RoboDK station: robodkproject048037074.rdk

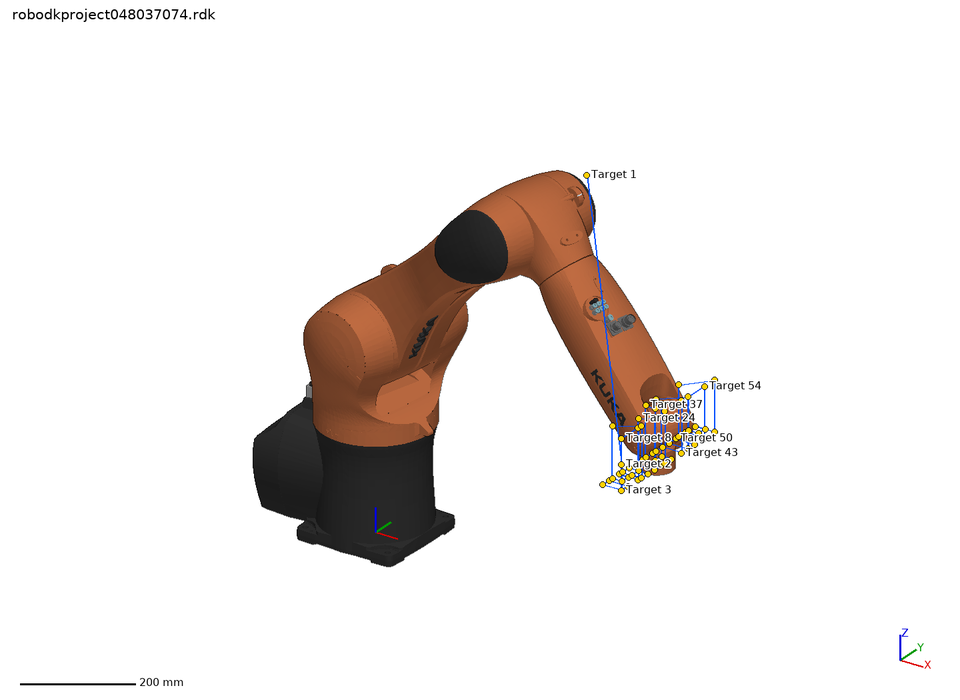
[picture v0: the station drawn from its stored meshes, robots at their saved joint values, targets as dots, program paths as lines]
Station robodkproject048037074 (saved by RoboDK 5.9.4). Poses are relative to the parent item; angles as X-Y-Z fixed-axis rotations.
  - frame KUKA KR 6 R900 sixx Base at (0, 0, 0) mm
    - robot KUKA KR 6 R900 sixx: 6 axes, payload 6 kg, reach 901 mm, repeatability 0.03 mm, weight 52 kg
        modified DH rows (alpha deg, a mm, theta deg, d mm): 0, 0, 0, 400; -90, 25, 0, 0; 0, 455, -90, 0; -90, 35, 0, 420; 90, 0, 0, 0; -90, 0, 180, 80
        joint limits [-170, -190, -120, -185, -120, -350] to [170, 45, 156, 185, 120, 350]; home [0, -90, 90, 0, 0, 0]; saved at [8.973, -42.929, 89.308, 0, 43.621, 8.973]
    - target Target 1 (Cartesian target) at (445, 0, 810) mm, rotated rx 180 ry 0 rz -180 deg; joints [0, -90, 90, 0, 90, 0] of KUKA KR 6 R900 sixx
    - target Target 2 (Cartesian target) at (665, -210, 400) mm, rotated rx 180 ry 0 rz -180 deg; joints [17.526, -44.432, 83.664, 0, 50.767, 17.526] of KUKA KR 6 R900 sixx
    - target Target 3 (Cartesian target) at (665, -210, 350) mm, rotated rx 180 ry 0 rz 180 deg; joints [17.526, -40.592, 84.501, 0, 46.092, 17.526] of KUKA KR 6 R900 sixx
    - target Target 4 (Cartesian target) at (625, -210, 350) mm, rotated rx 180 ry 0 rz -180 deg; joints [18.572, -44.227, 91.979, 0, 42.249, 18.572] of KUKA KR 6 R900 sixx
    - target Target 5 (Cartesian target) at (625, -190, 350) mm, rotated rx 180 ry 0 rz -180 deg; joints [16.909, -44.787, 93.129, 0, 41.657, 16.909] of KUKA KR 6 R900 sixx
    - target Target 6 (Cartesian target) at (665, -190, 350) mm, rotated rx 180 ry 0 rz -180 deg; joints [15.945, -41.161, 85.669, 0, 45.491, 15.945] of KUKA KR 6 R900 sixx
    - target Target 7 (Cartesian target) at (665, -210, 350) mm, rotated rx 180 ry 0 rz 180 deg; joints [17.526, -40.592, 84.501, 0, 46.092, 17.526] of KUKA KR 6 R900 sixx
    - target Target 8 (Cartesian target) at (665, -210, 450) mm, rotated rx 180 ry 0 rz 180 deg; joints [17.526, -47.839, 82.061, 0, 55.777, 17.526] of KUKA KR 6 R900 sixx
    - target Target 9 (Cartesian target) at (665, -160, 450) mm, rotated rx 180 ry 0 rz -180 deg; joints [13.528, -49.327, 84.778, 0, 54.549, 13.528] of KUKA KR 6 R900 sixx
    - target Target 10 (Cartesian target) at (665, -160, 350) mm, rotated rx 180 ry 0 rz -180 deg; joints [13.528, -41.903, 87.197, 0, 44.706, 13.528] of KUKA KR 6 R900 sixx
    - target Target 11 (Cartesian target) at (625, -160, 350) mm, rotated rx 180 ry 0 rz -180 deg; joints [14.359, -45.52, 94.638, 0, 40.882, 14.359] of KUKA KR 6 R900 sixx
    - target Target 12 (Cartesian target) at (645, -160, 350) mm, rotated rx 180 ry 0 rz -180 deg; joints [13.932, -43.745, 90.985, 0, 42.759, 13.932] of KUKA KR 6 R900 sixx
    - target Target 13 (Cartesian target) at (645, -180, 350) mm, rotated rx 180 ry 0 rz -180 deg; joints [15.593, -43.268, 90.005, 0, 43.263, 15.593] of KUKA KR 6 R900 sixx
    - target Target 14 (Cartesian target) at (625, -180, 350) mm, rotated rx 180 ry 0 rz -180 deg; joints [16.066, -45.045, 93.661, 0, 41.384, 16.066] of KUKA KR 6 R900 sixx
    - target Target 15 (Cartesian target) at (625, -180, 450) mm, rotated rx 180 ry 0 rz -180 deg; joints [16.066, -52.933, 91.269, 0, 51.664, 16.066] of KUKA KR 6 R900 sixx
    - target Target 16 (Cartesian target) at (665, -150, 450) mm, rotated rx 180 ry 0 rz -180 deg; joints [12.711, -49.576, 85.231, 0, 54.345, 12.711] of KUKA KR 6 R900 sixx
    - target Target 17 (Cartesian target) at (665, -150, 350) mm, rotated rx 180 ry 0 rz -180 deg; joints [12.711, -42.122, 87.647, 0, 44.475, 12.711] of KUKA KR 6 R900 sixx
    - target Target 18 (Cartesian target) at (665, -130, 350) mm, rotated rx 180 ry 0 rz -180 deg; joints [11.061, -42.516, 88.458, 0, 44.058, 11.061] of KUKA KR 6 R900 sixx
    - target Target 19 (Cartesian target) at (625, -130, 350) mm, rotated rx 180 ry 0 rz 180 deg; joints [11.75, -46.127, 95.887, 0, 40.24, 11.75] of KUKA KR 6 R900 sixx
    - target Target 20 (Cartesian target) at (625, -150, 350) mm, rotated rx 180 ry 0 rz -180 deg; joints [13.496, -45.736, 95.083, 0, 40.653, 13.496] of KUKA KR 6 R900 sixx
    - target Target 21 (Cartesian target) at (665, -150, 350) mm, rotated rx 180 ry 0 rz -180 deg; joints [12.711, -42.122, 87.647, 0, 44.475, 12.711] of KUKA KR 6 R900 sixx
    - target Target 22 (Cartesian target) at (645, -150, 350) mm, rotated rx 180 ry 0 rz -180 deg; joints [13.092, -43.962, 91.432, 0, 42.53, 13.092] of KUKA KR 6 R900 sixx
    - target Target 23 (Cartesian target) at (645, -130, 350) mm, rotated rx 180 ry 0 rz -180 deg; joints [11.395, -44.353, 92.238, 0, 42.115, 11.395] of KUKA KR 6 R900 sixx
    - target Target 24 (Cartesian target) at (645, -130, 450) mm, rotated rx 180 ry 0 rz -180 deg; joints [11.395, -52.134, 89.842, 0, 52.292, 11.395] of KUKA KR 6 R900 sixx
    - target Target 25 (Cartesian target) at (665, -110, 450) mm, rotated rx 180 ry 0 rz -180 deg; joints [9.392, -50.412, 86.745, 0, 53.667, 9.392] of KUKA KR 6 R900 sixx
    - target Target 26 (Cartesian target) at (665, -110, 350) mm, rotated rx 180 ry 0 rz -180 deg; joints [9.392, -42.854, 89.153, 0, 43.701, 9.392] of KUKA KR 6 R900 sixx
    - target Target 27 (Cartesian target) at (665, -90, 350) mm, rotated rx 180 ry 0 rz -180 deg; joints [7.707, -43.135, 89.731, 0, 43.404, 7.707] of KUKA KR 6 R900 sixx
    - target Target 28 (Cartesian target) at (625, -90, 350) mm, rotated rx 180 ry 0 rz -180 deg; joints [8.194, -46.74, 97.15, 0, 39.59, 8.194] of KUKA KR 6 R900 sixx
    - target Target 29 (Cartesian target) at (625, -110, 350) mm, rotated rx 180 ry 0 rz -180 deg; joints [9.982, -46.461, 96.576, 0, 39.885, 9.982] of KUKA KR 6 R900 sixx
    - target Target 30 (Cartesian target) at (665, -110, 350) mm, rotated rx 180 ry 0 rz -180 deg; joints [9.392, -42.854, 89.153, 0, 43.701, 9.392] of KUKA KR 6 R900 sixx
    - target Target 31 (Cartesian target) at (665, -110, 450) mm, rotated rx 180 ry 0 rz -180 deg; joints [9.392, -50.412, 86.745, 0, 53.667, 9.392] of KUKA KR 6 R900 sixx
    - target Target 32 (Cartesian target) at (665, -80, 450) mm, rotated rx 180 ry 0 rz -180 deg; joints [6.86, -50.87, 87.572, 0, 53.298, 6.86] of KUKA KR 6 R900 sixx
    - target Target 33 (Cartesian target) at (665, -80, 350) mm, rotated rx 180 ry 0 rz -180 deg; joints [6.86, -43.254, 89.976, 0, 43.278, 6.86] of KUKA KR 6 R900 sixx
    - target Target 34 (Cartesian target) at (665, -60, 350) mm, rotated rx 180 ry 0 rz -180 deg; joints [5.156, -43.45, 90.38, 0, 43.07, 5.156] of KUKA KR 6 R900 sixx
    - target Target 35 (Cartesian target) at (625, -60, 350) mm, rotated rx 180 ry 0 rz -180 deg; joints [5.484, -47.054, 97.797, 0, 39.258, 5.484] of KUKA KR 6 R900 sixx
    - target Target 36 (Cartesian target) at (625, -80, 350) mm, rotated rx 180 ry 0 rz -180 deg; joints [7.294, -46.859, 97.395, 0, 39.464, 7.294] of KUKA KR 6 R900 sixx
    - target Target 37 (Cartesian target) at (625, -80, 450) mm, rotated rx 180 ry 0 rz -180 deg; joints [7.294, -55.044, 95.003, 0, 50.041, 7.294] of KUKA KR 6 R900 sixx
    - target Target 38 (Cartesian target) at (645, -80, 450) mm, rotated rx 180 ry 0 rz -180 deg; joints [7.07, -52.982, 91.355, 0, 51.626, 7.07] of KUKA KR 6 R900 sixx
    - target Target 39 (Cartesian target) at (645, -80, 350) mm, rotated rx 180 ry 0 rz -180 deg; joints [7.07, -45.087, 93.747, 0, 41.34, 7.07] of KUKA KR 6 R900 sixx
    - target Target 40 (Cartesian target) at (645, -60, 350) mm, rotated rx 180 ry 0 rz -180 deg; joints [5.315, -45.282, 94.15, 0, 41.133, 5.315] of KUKA KR 6 R900 sixx
    - target Target 41 (Cartesian target) at (645, -60, 450) mm, rotated rx 180 ry 0 rz -180 deg; joints [5.315, -53.208, 91.758, 0, 51.45, 5.315] of KUKA KR 6 R900 sixx
    - target Target 42 (Cartesian target) at (665, -30, 450) mm, rotated rx 180 ry 0 rz -180 deg; joints [2.583, -51.313, 88.369, 0, 52.944, 2.583] of KUKA KR 6 R900 sixx
    - target Target 43 (Cartesian target) at (665, -30, 350) mm, rotated rx 180 ry 0 rz -180 deg; joints [2.583, -43.64, 90.769, 0, 42.87, 2.583] of KUKA KR 6 R900 sixx
    - target Target 44 (Cartesian target) at (625, -30, 350) mm, rotated rx 180 ry 0 rz -180 deg; joints [2.748, -47.243, 98.185, 0, 39.058, 2.748] of KUKA KR 6 R900 sixx
    - target Target 45 (Cartesian target) at (625, -50, 350) mm, rotated rx 180 ry 0 rz -180 deg; joints [4.574, -47.131, 97.955, 0, 39.176, 4.574] of KUKA KR 6 R900 sixx
    - target Target 46 (Cartesian target) at (625, -50, 450) mm, rotated rx 180 ry 0 rz -180 deg; joints [4.574, -55.363, 95.563, 0, 49.8, 4.574] of KUKA KR 6 R900 sixx
    - target Target 47 (Cartesian target) at (665, -10, 450) mm, rotated rx 180 ry 0 rz -180 deg; joints [0.862, -51.377, 88.485, 0, 52.893, 0.862] of KUKA KR 6 R900 sixx
    - target Target 48 (Cartesian target) at (665, -10, 350) mm, rotated rx 180 ry 0 rz -180 deg; joints [0.862, -43.696, 90.885, 0, 42.811, 0.862] of KUKA KR 6 R900 sixx
    - target Target 49 (Cartesian target) at (665, 10, 350) mm, rotated rx 180 ry 0 rz -180 deg; joints [-0.862, -43.696, 90.885, 0, 42.811, -0.862] of KUKA KR 6 R900 sixx
    - target Target 50 (Cartesian target) at (625, 10, 350) mm, rotated rx 180 ry 0 rz -180 deg; joints [-0.917, -47.299, 98.3, 0, 38.999, -0.917] of KUKA KR 6 R900 sixx
    - target Target 51 (Cartesian target) at (625, -10, 350) mm, rotated rx 180 ry 0 rz -180 deg; joints [0.917, -47.299, 98.3, 0, 38.999, 0.917] of KUKA KR 6 R900 sixx
    - target Target 52 (Cartesian target) at (665, -10, 350) mm, rotated rx 180 ry 0 rz -180 deg; joints [0.862, -43.696, 90.885, 0, 42.811, 0.862] of KUKA KR 6 R900 sixx
    - target Target 53 (Cartesian target) at (665, -10, 450) mm, rotated rx 180 ry 0 rz -180 deg; joints [0.862, -51.377, 88.485, 0, 52.893, 0.862] of KUKA KR 6 R900 sixx
    - target Target 54 (Cartesian target) at (665, 40, 450) mm, rotated rx 180 ry 0 rz -180 deg; joints [-3.442, -51.256, 88.268, 0, 52.989, -3.442] of KUKA KR 6 R900 sixx
    - target Target 55 (Cartesian target) at (665, 40, 350) mm, rotated rx 180 ry 0 rz -180 deg; joints [-3.442, -43.59, 90.668, 0, 42.922, -3.442] of KUKA KR 6 R900 sixx
    - target Target 56 (Cartesian target) at (625, 40, 350) mm, rotated rx 180 ry 0 rz -180 deg; joints [-3.662, -47.194, 98.084, 0, 39.11, -3.662] of KUKA KR 6 R900 sixx
    - target Target 57 (Cartesian target) at (625, 20, 350) mm, rotated rx 180 ry 0 rz -180 deg; joints [-1.833, -47.278, 98.257, 0, 39.021, -1.833] of KUKA KR 6 R900 sixx
    - target Target 58 (Cartesian target) at (625, 20, 450) mm, rotated rx 180 ry 0 rz -180 deg; joints [-1.833, -55.535, 95.864, 0, 49.671, -1.833] of KUKA KR 6 R900 sixx
    - target Target 59 (Cartesian target) at (665, 70, 450) mm, rotated rx 180 ry 0 rz -180 deg; joints [-6.009, -50.991, 87.79, 0, 53.201, -6.009] of KUKA KR 6 R900 sixx
    - target Target 60 (Cartesian target) at (665, 70, 350) mm, rotated rx 180 ry 0 rz -180 deg; joints [-6.009, -43.359, 90.192, 0, 43.167, -6.009] of KUKA KR 6 R900 sixx
    - target Target 61 (Cartesian target) at (625, 70, 350) mm, rotated rx 180 ry 0 rz -180 deg; joints [-6.39, -46.964, 97.61, 0, 39.354, -6.39] of KUKA KR 6 R900 sixx
    - target Target 62 (Cartesian target) at (645, 70, 350) mm, rotated rx 180 ry 0 rz -180 deg; joints [-6.194, -45.192, 93.963, 0, 41.229, -6.194] of KUKA KR 6 R900 sixx
    - target Target 63 (Cartesian target) at (645, 50, 350) mm, rotated rx 180 ry 0 rz -180 deg; joints [-4.433, -45.359, 94.308, 0, 41.052, -4.433] of KUKA KR 6 R900 sixx
    - target Target 64 (Cartesian target) at (625, 50, 350) mm, rotated rx 180 ry 0 rz -180 deg; joints [-4.574, -47.131, 97.955, 0, 39.176, -4.574] of KUKA KR 6 R900 sixx
  - program meca315yg (65 instructions, listed below)
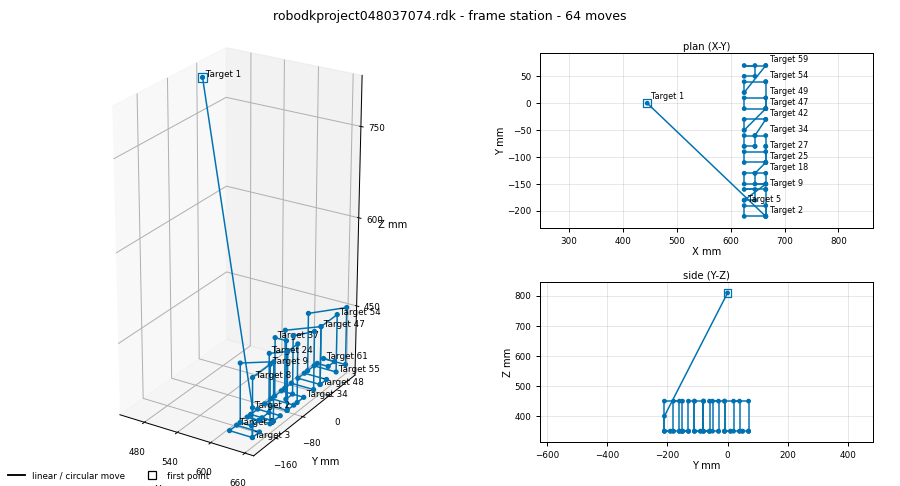
[picture p0: tool path of robodkproject048037074.rdk in frame station, 64 of 64 moves have a stored position in this frame; points joined in program order, loops and branches not executed]

--- program meca315yg (robot KUKA KR 6 R900 sixx) ---
  Set Ref.: KUKA KR 6 R900 sixx Base
  MoveJ (Target 1)
  MoveL (Target 2)
  MoveL (Target 3)
  MoveL (Target 4)
  MoveL (Target 5)
  MoveL (Target 6)
  MoveL (Target 7)
  MoveL (Target 8)
  MoveL (Target 9)
  MoveL (Target 10)
  MoveL (Target 11)
  MoveL (Target 12)
  MoveL (Target 13)
  MoveL (Target 14)
  MoveL (Target 15)
  MoveL (Target 16)
  MoveL (Target 17)
  MoveL (Target 18)
  MoveL (Target 19)
  MoveL (Target 20)
  MoveL (Target 21)
  MoveL (Target 22)
  MoveL (Target 23)
  MoveL (Target 24)
  MoveL (Target 25)
  MoveL (Target 26)
  MoveL (Target 27)
  MoveL (Target 28)
  MoveL (Target 29)
  MoveL (Target 30)
  MoveL (Target 31)
  MoveL (Target 32)
  MoveL (Target 33)
  MoveL (Target 34)
  MoveL (Target 35)
  MoveL (Target 36)
  MoveL (Target 37)
  MoveL (Target 38)
  MoveL (Target 39)
  MoveL (Target 40)
  MoveL (Target 41)
  MoveL (Target 42)
  MoveL (Target 43)
  MoveL (Target 44)
  MoveL (Target 45)
  MoveL (Target 46)
  MoveL (Target 47)
  MoveL (Target 48)
  MoveL (Target 49)
  MoveL (Target 50)
  MoveL (Target 51)
  MoveL (Target 52)
  MoveL (Target 53)
  MoveL (Target 54)
  MoveL (Target 55)
  MoveL (Target 56)
  MoveL (Target 57)
  MoveL (Target 58)
  MoveL (Target 59)
  MoveL (Target 60)
  MoveL (Target 61)
  MoveL (Target 62)
  MoveL (Target 63)
  MoveL (Target 64)
